(* PLC project Generated.project, CODESYS CODESYS V3.5 SP19 Patch 1 *)
(* stored: creationDateTime 2026-09-06T13:00:42.487648, modificationDateTime 2026-09-06T13:00:42.487648 *)

(* ======================================================================= ST_TraceWinch - Trace de blocage terrain d'un treuil M1/M2 ----------------------------------------------------------------------- Role : Publier au technicien une vue consolidee "pourquoi l'axe ne bouge pas" : permis effectifs par sens, source du SafeStop/coupure, cause de blocage priorisee et horodatee. Producteur unique : PRG_04_Treuils_Benne (#8bis) - 1 instance par axe (TraceM1 / TraceM2 au sein de ST_WinchInterPrg). Consommateur : FB_TroubleshootingView (pure recopie -> GVL_Troubleshooting). Lecture seule - aucun calcul de commande n'en depend. BlockReasonTimestamp : ms depuis demarrage PLC (TIME()), latched au dernier changement de BlockReason (1 scan, memoire). Doc metier : DOC/AF/AF_Partie-14_Fonction_Troubleshooting_v1.4.md ======================================================================= *)
TYPE ST_TraceWinch : STRUCT
  DescendPermitEffective : BOOL;  (* Permis effectifs par sens (reflet exact des permis appliques au mouvement) Descente effectivement permise (EffectivePermit*_Descend) *)
  AscentPermitEffective : BOOL;  (* Montee effectivement permise (EffectivePermit*_Ascent) *)
  AscentPermitApplied : BOOL;  (* Permis effectivement transmis a la barriere finale *)
  DescendPermitApplied : BOOL;  (* Permis effectivement transmis a la barriere finale *)
  FinalPermitBlocked : BOOL;  (* Demande presente mais refusee par le permis final *)
  SafeStopActive : BOOL;  (* Source de SafeStop / coupure - pour distinguer l'origine du blocage SafeStop effectif applique (SafeStop*_Active) *)
  SafeStopSourceSafety : BOOL;  (* SafeStop issu de FB_Safety_Winch (defaut safety) *)
  SafeStopSourceInput : BOOL;  (* SafeStop issu du module d'entree / homing / slip benne *)
  SafeStopSourceSync : BOOL;  (* SafeStop issu de la synchro M1/M2 (couplage anti-telescopage) *)
  PowerCutOffActive : BOOL;  (* Coupure puissance amont active (instSafetyWinch.PowerCutOff) *)
  Inhibited : BOOL;  (* Axe neutralise (Mode=DISABLE ou InhibitMx) *)
  FinalInterlockError : BOOL;  (* Barriere finale (fin de course mecanique / frein / redemarrage) Defaut barriere finale (frein / redemarrage) *)
  FinalInterlockReason : E_WinchFinalInterlockReason;  (* Cause barriere finale memorisee *)
  BlockReason : E_WinchTraceBlockReason;  (* Cause de blocage priorisee + horodatage Cause de blocage prioritaire *)
  BlockReasonTimestamp : UDINT;  (* ms depuis demarrage PLC (TIME()) - dernier changement de BlockReason *)
  StepNumber : INT;  (* Palier de vitesse actif (WinchState.StepNumber) *)
END_STRUCT;
END_TYPE

(* values of E_WinchFinalInterlockReason: NONE: Aucun blocage actif; BRAKE_COMMAND_NOT_CONFIRMED: Absence confirmation ouverture frein > 500ms; RESTART_INHIBITED: Inhibition redemarrage actif; SENSE_DROP_TIMEOUT: T_max §3bis depasse sans confirmation retombee (AC7) *)

{attribute 'qualified_only'}
{attribute 'strict'}
TYPE E_WinchFinalInterlockReason : (NONE := 0, BRAKE_COMMAND_NOT_CONFIRMED := 1, RESTART_INHIBITED := 2, SENSE_DROP_TIMEOUT := 3);
END_TYPE

(* values of E_WinchTraceBlockReason: NONE: Aucun blocage - au moins un sens effectivement permis; POWER_CUTOFF: Coupure puissance amont (instSafetyWinch.PowerCutOff) - priorite max; AXIS_DISABLED: Axe neutralise (Mode=DISABLE ou InhibitMx -> Enable FALSE); SAFESTOP: SafeStop effectif (rampe rapide demandee); SAFETY_FAULT: Defaut safety latched (FB_Safety_Winch.Fault.Error); SAFETY_PERMIT_MISSING: Aucun sens ne delivre de permit safety (limite / mou de cable / homing); PROCESS_PERMIT_MISSING: Permit process absent (benne / fond Kobold / limite legale / extraction); COUPLING_BLOCKED: Couplage synchro anti-telescopage (l'autre axe bloque); WINCH_FAULT: Defaut treuil latched (FB_Winch.Fault.Error); FINAL_INTERLOCK_BLOCKED: Barriere finale en defaut (frein / redemarrage) *)

{attribute 'qualified_only'}
{attribute 'strict'}
TYPE E_WinchTraceBlockReason : (NONE := 0, POWER_CUTOFF := 1, AXIS_DISABLED := 2, SAFESTOP := 3, SAFETY_FAULT := 4, SAFETY_PERMIT_MISSING := 5, PROCESS_PERMIT_MISSING := 6, COUPLING_BLOCKED := 7, WINCH_FAULT := 8, FINAL_INTERLOCK_BLOCKED := 9);
END_TYPE
